FUNCTION_BLOCK FB_MQTTCommunication
VAR_INPUT
END_VAR
VAR_OUTPUT
END_VAR
VAR
	GetHostName:		FB_GetHostName;
	HostName: 			STRING(255);
    bSetParameter:		BOOL := FALSE;
    bConnect:			BOOL := FALSE;
    (* received message *)
	bSubscribed: 		BOOL;
	sTopicSub: 			STRING(255) := 'STELLA1/Telescope/SET';
	{attribute 'TcEncoding':='UTF-8'}
	sTopicRcv: 			STRING(255);
	{attribute 'TcEncoding':='UTF-8'}
	fbMessageQueue:		FB_IotMqttMessageQueue;
    fbMessage:			FB_IotMqttMessage;
	fbMqttClient:		FB_IotMqttClient;
	sPayloadRcv: 		STRING;
	influxMessage:		FB_InfluxMessage;
	measurement, 
	parameter, 
	value:		STRING(255);
END_VAR

(*
MQTT Communication section

Source:
https://infosys.beckhoff.com/english.php?content=../content/1033/tf6701_tc3_iot_communication_mqtt/3518541195.html&id=

*)
IF HostName='' THEN
	GetHostName.bExecute := TRUE;
ELSE
	GetHostName.bExecute := FALSE;
	bSetParameter := TRUE;
END_IF

GetHostName(sHostName => HostName);

// set the parameters once
IF bSetParameter THEN
    bSetParameter               := FALSE;
    fbMqttClient.sHostName      := 'sky.stella.iac.es';
    fbMqttClient.nHostPort      := 1883;
    fbMqttClient.sClientId      := HostName; 
    fbMqttClient.sTopicPrefix   := ''; 
	fbMqttClient.nKeepAlive     := 60; 
    fbMqttClient.ipMessageQueue := fbMessageQueue;
	bConnect := TRUE;
END_IF

// connect to the client
IF NOT fbMqttClient.bConnected THEN
;
END_IF

fbMqttClient.Execute(bConnect);
	
IF fbMqttClient.bConnected THEN
    IF NOT bSubscribed THEN
        bSubscribed := fbMqttClient.Subscribe(sTopic:=sTopicSub, 
												eQoS:=TcIotMqttQos.AtMostOnceDelivery);
    END_IF
END_IF

// receive queued messages
IF fbMessageQueue.nQueuedMessages > 0 THEN
    IF fbMessageQueue.Dequeue(fbMessage:=fbMessage) THEN
        fbMessage.GetTopic(pTopic:=ADR(sTopicRcv), nTopicSize:=SIZEOF(sTopicRcv) );
        fbMessage.GetPayload(pPayload:=ADR(sPayloadRcv), nPayloadSize:=SIZEOF(sPayloadRcv), bSetNullTermination:=TRUE);
		ADSLOGSTR( ADSLOG_MSGTYPE_HINT OR ADSLOG_MSGTYPE_LOG, 'MQTT %s', sPayloadRcv);
		IF sTopicRcv = sTopicSub THEN
			influxMessage(  sPayload := sPayloadRcv, measurement => measurement, parameter => parameter, value => value);
			IF NOT PendantControl.manual AND measurement = 'command' THEN
				IF parameter = 'power' THEN
					TelescopeControl.power := STRING_TO_BOOL(value);
				ELSIF parameter = 'park' THEN
					TelescopeControl.park := STRING_TO_BOOL(value);
				ELSIF parameter = 'gohome' THEN
					TelescopeControl.gohome := STRING_TO_BOOL(value);
				ELSIF parameter = 'track' THEN
					TelescopeControl.track := STRING_TO_BOOL(value);
				ELSIF parameter = 'goto' THEN
					TelescopeControl.goto := STRING_TO_BOOL(value);
				ELSIF parameter = 'slew' THEN
					TelescopeControl.slew := STRING_TO_BOOL(value);
				ELSIF parameter = 'stop' THEN
					TelescopeControl.stop := STRING_TO_BOOL(value);
				ELSIF parameter = 'reset' THEN
					TelescopeControl.reset := STRING_TO_BOOL(value);
				ELSIF parameter = 'masterreset' THEN
					ElevationControl.bSoEReset := STRING_TO_BOOL(value);
					AzimuthElevationControl.bSoEReset := STRING_TO_BOOL(value);
					DerotatorControl.bSoEReset := STRING_TO_BOOL(value);
				ELSIF parameter = 'nasmyth' THEN
					NasmythControl.left := STRING_TO_USINT(value) = 1;
					NasmythControl.right := STRING_TO_USINT(value) = 2;
				ELSIF parameter = 'rightascension' THEN
					TelescopeControl.track := FALSE;
					TelescopeControl.rightascension := STRING_TO_LREAL(value);
				ELSIF parameter = 'declination' THEN
					TelescopeControl.track := FALSE;
					TelescopeControl.declination := STRING_TO_LREAL(value);
				ELSIF parameter = 'elevation' THEN
					TelescopeControl.elevation := STRING_TO_LREAL(value);
				ELSIF parameter = 'azimuth' THEN
					TelescopeControl.azimuth := STRING_TO_LREAL(value);
				ELSIF parameter = 'focus' THEN
					FocusControl.position := STRING_TO_LREAL(value);
				ELSIF parameter = 'filter' THEN
					FilterWheelControl.filter_position := STRING_TO_USINT(value);
				ELSIF parameter = 'derotator' THEN
					TelescopeControl.track := FALSE;
					TelescopeControl.derotator_offset := STRING_TO_LREAL(value);
				ELSIF parameter = 'elevationoffset' THEN
					TelescopeControl.elevation_offset := STRING_TO_LREAL(value);
				ELSIF parameter = 'azimuthoffset' THEN
					TelescopeControl.azimuth_offset := STRING_TO_LREAL(value);
				ELSIF parameter = 'derotatoroffset' THEN
					TelescopeControl.derotator_offset := STRING_TO_LREAL(value);ELSE
					ADSLOGSTR( ADSLOG_MSGTYPE_WARN OR ADSLOG_MSGTYPE_LOG, 'MQTT not understood %s', sPayloadRcv);
				END_IF
			END_IF // measurement
		END_IF // Topic
		sPayloadRcv := '';
    END_IF // Dequeue
END_IF

PROPERTY Error : BOOL
GET
Error := fbMqttClient.bError;
END_GET
END_PROPERTY

METHOD Publish : BOOL
VAR_INPUT
	domain: 	STRING(255) := 'environment';
	location: 	STRING(255) := 'roof';
	parameter:	STRING(255);
	value:		STRING(255);
END_VAR
VAR
	sPayloadPub: STRING(255) := '';
	fbFormat:	FB_FormatString;
	bError:		BOOL;
	nErrID: UDINT;
	retain_message:		BOOL := FALSE;
END_VAR
//sPayloadPub := 'environment,location=roof,host=CX-4E6032 ';
fbFormat( sFormat := '%s,location=%s,host=%s %s=%s', 
			arg1 := F_STRING(domain), 
			arg2 := F_STRING(location), 
			arg3 := F_STRING(HostName),
			arg4 := F_STRING(parameter),
			arg5 := F_STRING(value),
 
			sOut => sPayloadPub,
			bError => bError, 
			nErrID => nErrID );
// retain message if value is boolean
retain_message := value = 'TRUE' OR value = 'FALSE';

Publish := fbMqttClient.Publish(	
				sTopic:= 'STELLA1/Telemetry', 
				pPayload:= ADR(sPayloadPub), 
				nPayloadSize:= LEN2(ADR(sPayloadPub)),
				eQoS:= TcIotMqttQos.AtMostOnceDelivery,
				bRetain:= retain_message, 
				bQueue:= FALSE );
END_METHOD

METHOD PublishLog : BOOL
VAR_INPUT
	level: 	STRING(255) := 'INFO';
	message:	STRING(255);
	
END_VAR
VAR
	sPayloadPub: STRING(255) := '';
	fbFormat:	FB_FormatString;
	bError:		BOOL;
	nErrID: UDINT;
END_VAR
VAR_OUTPUT
	published: BOOL;
END_VAR
//sPayloadPub := 'environment,location=roof,host=CX-4E6032 ';
fbFormat( sFormat := 'log,host=%s,level=%s message="%s"', 
			arg1 := F_STRING(HostName), 
			arg2 := F_STRING(level), 
			arg3 := F_STRING(message),
 
			sOut => sPayloadPub,
			bError => bError, 
			nErrID => nErrID );

published := fbMqttClient.Publish(	
				sTopic:= 'STELLA1/Log', 
				pPayload:= ADR(sPayloadPub), 
				nPayloadSize:= LEN2(ADR(sPayloadPub)),
				eQoS:= TcIotMqttQos.AtMostOnceDelivery,
				bRetain:= FALSE, 
				bQueue:= FALSE );
END_METHOD

END_FUNCTION_BLOCK

(* stored: Version 1.1.0.1, ProductVersion 3.1.4024.9
   POU FB_MQTTCommunication: Id {5f9ef57f-1a43-46d5-9870-b05542416a37}, SpecialFunc None
   Property Error: Id {78d1d012-baaf-423e-a194-3780c6f6dc78}
   Get Get: Id {06797971-03f0-42f5-8ce7-317a6cd32c60}
   Method Publish: Id {cdbc3347-8b58-489a-94fe-8e8502587296}
   Method PublishLog: Id {e0ebb0b3-f1b8-4a54-a57a-d713d9f93164} *)
